TYPE FsT_PlcAppInfo : PlcAppSystemInfo; END_TYPE

(* stored: Version 1.1.0.1, ProductVersion 3.1.4024.4
   DUT FsT_PlcAppInfo: Id {3f4ae9eb-f05e-4973-9ce1-927207e78951} *)
